(* Schneider Machine Expert - Basic project Project_kopchennya, file version 2.9.0.0 *)
(* ProjectInformations: Name=Project_kopchennya *)

HARDWARE
  Cpu 0: TM221CE24T
  ModuleExtensionObject 0: TM2ALM3LT
  EthernetConfiguration: NetworkName=M221, IpAllocationMode=FixedAddress, IpAddress=0.0.0.0, SubnetMask=0.0.0.0
  SerialLineConfiguration: Baud=Baud19200, Parity=ParityEven, DataBits=DataBits8, StopBits=StopBits1, PhysicalMedium=PhysicalMediumRs485, TransmissionMode=TransmissionModeModbusRtu, SlaveId=1, Addressing=SlaveAddressing
  MastTask: UsePeriodScanMode=false, PeriodScan=100
  FastTask: Period=255
  CpuBehavior: StartingMode=StartAsPreviousState, AutoSaveRamOnEeprom=true, WatchdogPeriod=250

SYMBOLS  (address, symbol, comment, settings)
  %M0       PHASE_0  "Memory Phase 0"
  %M1       PHASE_1  "Memory Phase 1"
  %M2       PHASE_2  "Memory Phase 2"
  %M3       PHASE_3  "Memory Phase 3"
  %M4       PHASE_4  "Memory Phase 4"
  %TM0        [Type=TP, Preset=30, Base=OneSecond]
  %TM1        [Preset=30, Base=OneSecond]
  %TM2        [Type=TP, Preset=30, Base=OneSecond]
  %TM3        [Preset=30, Base=OneSecond]
  %I0.0     BUTTON_STOP  "Button "STOP/RESET""
  %I0.1     BUTTON_START  "Button "START""
  %I0.2     BUTTON_PAUSE  "Button "PAUSE""
  %I0.3     SENSOR_DOOR  "Input Sensor Door"
  %I0.4     SENSOR_PHOTO  "Input Photo Sensor"
  %Q0.0     FAN  "Fan"
  %Q0.1     HEATER  "Air Heater"
  %Q0.2     SMOKE_GENERATOR  "Smoke Generator"
  %Q0.3     LED_STOP  "LED STOP"
  %Q0.4     LED_PHASE_1  "LED Phase 1"
  %Q0.5     LED_PHASE_2  "LED Phase 2"
  %Q0.6     LED_PHASE_3  "LED Phase 3"
  %Q0.7     LED_PHASE_4  "LED Phase 4"
  %IW0.0    SENSOR_HUM  "Sensor Humidity"  [Type=Type_0_10V, Scope=Scope_Normal, Minimum=0, Maximum=1000]
  %IW1.0    SENSOR_TEMP  "Sensor Temperature"  [Type=Type_PT100, Scope=Scope_Celsius, Minimum=-1000, Maximum=5000]
  %QW1.0    CONTROL_DAMPER  "Control Damper"  [Type=Type_0_10V, Scope=Scope_Customized, Minimum=0, Maximum=100]

POU New POU
  (* SectionNumber=1 *)

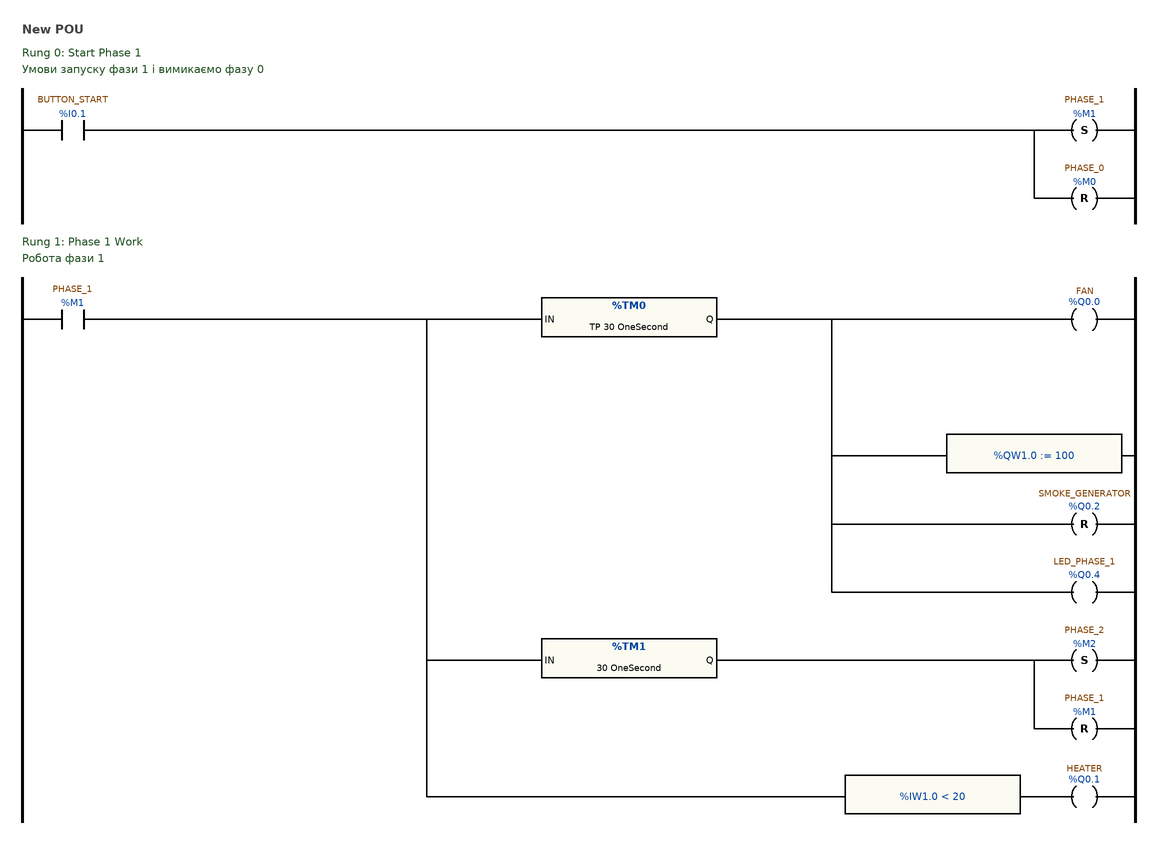

// Rung 0: Start Phase 1
// Умови запуску фази 1 і вимикаємо фазу 0
  LD %I0.1                (* BUTTON_START *)
  S %M1                   (* PHASE_1 *)
  R %M0                   (* PHASE_0 *)
  // as ST:
  //   IF BUTTON_START THEN PHASE_1 := TRUE; END_IF;
  //   IF BUTTON_START THEN PHASE_0 := FALSE; END_IF;

// Rung 1: Phase 1 Work
// Робота фази 1
  LD 1
  MULTIFB
  LD 1
  AND %M1                 (* PHASE_1 *)
  ST %MW2009:X0
  BLK %TM0
  LD %MW2009:X0
  IN
  OUT_BLK
  LD Q
  ST %Q0.0                (* FAN *)
  [ %QW1.0 := 100 ]       (* CONTROL_DAMPER *)
  R %Q0.2                 (* SMOKE_GENERATOR *)
  ST %Q0.4                (* LED_PHASE_1 *)
  END_BLK
  BLK %TM1
  LD %MW2009:X0
  IN
  OUT_BLK
  LD Q
  S %M2                   (* PHASE_2 *)
  R %M1                   (* PHASE_1 *)
  END_BLK
  LD %MW2009:X0
  AND [ %IW1.0 < 20 ]     (* SENSOR_TEMP *)
  ST %Q0.1                (* HEATER *)
  MULTIFB
  // as ST:
  //   %TM0(IN := PHASE_1);
  //   FAN := %TM0.Q;
  //   IF %TM0.Q THEN CONTROL_DAMPER := 100; END_IF;
  //   IF %TM0.Q THEN SMOKE_GENERATOR := FALSE; END_IF;
  //   LED_PHASE_1 := %TM0.Q;
  //   %TM1(IN := PHASE_1);
  //   IF %TM1.Q THEN PHASE_2 := TRUE; END_IF;
  //   _t1 := PHASE_1;
  //   IF %TM1.Q THEN PHASE_1 := FALSE; END_IF;
  //   HEATER := _t1 AND SENSOR_TEMP < 20;

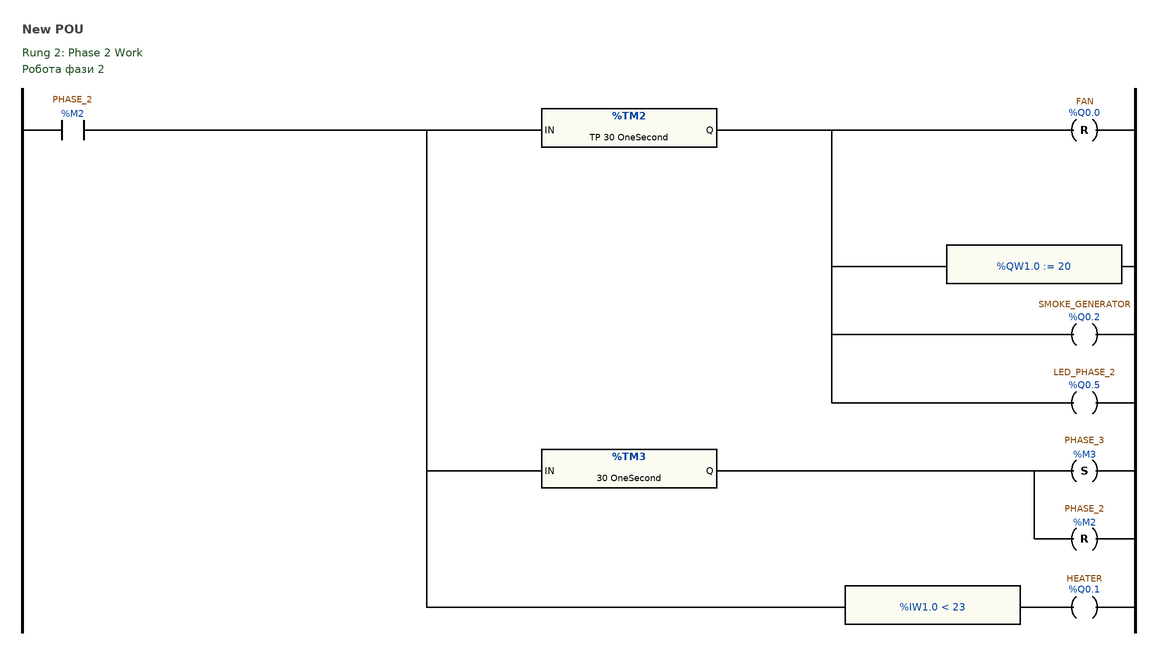

// Rung 2: Phase 2 Work
// Робота фази 2
  LD 1
  MULTIFB
  LD 1
  AND %M2                 (* PHASE_2 *)
  ST %MW2009:X0
  BLK %TM2
  LD %MW2009:X0
  IN
  OUT_BLK
  LD Q
  R %Q0.0                 (* FAN *)
  [ %QW1.0 := 20 ]        (* CONTROL_DAMPER *)
  ST %Q0.2                (* SMOKE_GENERATOR *)
  ST %Q0.5                (* LED_PHASE_2 *)
  END_BLK
  BLK %TM3
  LD %MW2009:X0
  IN
  OUT_BLK
  LD Q
  S %M3                   (* PHASE_3 *)
  R %M2                   (* PHASE_2 *)
  END_BLK
  LD %MW2009:X0
  AND [ %IW1.0 < 23 ]     (* SENSOR_TEMP *)
  ST %Q0.1                (* HEATER *)
  MULTIFB
  // as ST:
  //   %TM2(IN := PHASE_2);
  //   IF %TM2.Q THEN FAN := FALSE; END_IF;
  //   IF %TM2.Q THEN CONTROL_DAMPER := 20; END_IF;
  //   SMOKE_GENERATOR := %TM2.Q;
  //   LED_PHASE_2 := %TM2.Q;
  //   %TM3(IN := PHASE_2);
  //   IF %TM3.Q THEN PHASE_3 := TRUE; END_IF;
  //   _t1 := PHASE_2;
  //   IF %TM3.Q THEN PHASE_2 := FALSE; END_IF;
  //   HEATER := _t1 AND SENSOR_TEMP < 23;
